// Mitsubishi GX Works2 project: 카운터   PLC: Q02/Q02H

PROGRAM MAIN
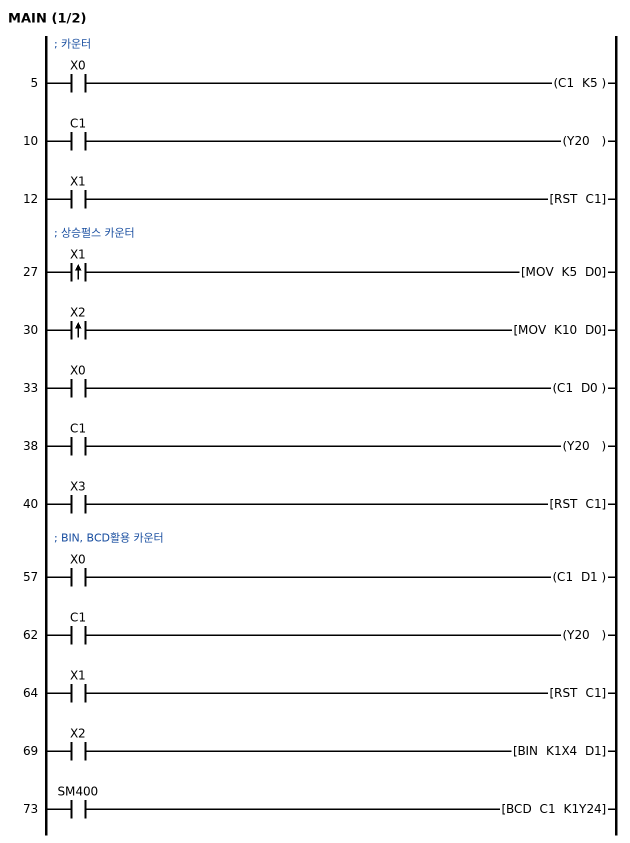
; 카운터
5     LD      X0
      OUT     C1 K5
10    LD      C1
      OUT     Y20
12    LD      X1
      RST     C1
; 상승펄스 카운터
27    LDP     X1
      MOV     K5 D0
30    LDP     X2
      MOV     K10 D0
33    LD      X0
      OUT     C1 D0
38    LD      C1
      OUT     Y20
40    LD      X3
      RST     C1
; BIN, BCD활용 카운터
57    LD      X0
      OUT     C1 D1
62    LD      C1
      OUT     Y20
64    LD      X1
      RST     C1
69    LD      X2
      BIN     K1X4 D1
73    LD      SM400
      BCD     C1 K1Y24
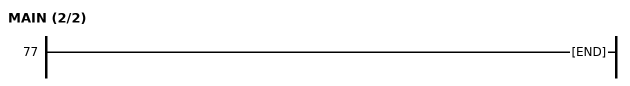
77    END
END_PROGRAM
